FUNCTION_BLOCK MainStation EXTENDS TcoCore.TcoObject
VAR
    counter : INT;

    testAxis : AxisIaiLibrary.AxisIAI(THIS^, AxisLimits := AxisStats.AxisLimitsRfid);

    enable                 : BOOL := TRUE;
    controllWithCommActive : BOOL := TRUE;
    //Link this for example in Global to IN/Out
    gateWayStatus      : AxisIaiLibrary.GatewayStatus;
    gateWayControl     : AxisIaiLibrary.GatewayControl;
    DriveToPlcTestAxis : AxisIaiLibrary.PlcIn;
    PlcToDriveTestAxis : AxisIaiLibrary.PlcOut;
END_VAR

counter := counter + 1;

IF (THIS^.counter MOD 13 = 0) THEN
    THIS^.Messenger.Info('opalalla').Pin();
END_IF

IF (THIS^.counter MOD 400 = 0) THEN
    THIS^.Messenger.Error('ich Poste').Pin();
END_IF

testAxis
(
    inEnabled        := enable
    , GateWayStatus  := gateWayStatus
    , GateWayControl := gateWayControl
    , DriveToPlc     := DriveToPlcTestAxis
    , PlcToDrive     := PlcToDriveTestAxis
);

gateWayControl.GatewayControl0.MON := controllWithCommActive;

END_FUNCTION_BLOCK

(* stored: Version 1.1.0.1, ProductVersion 3.1.4024.12
   POU MainStation: Id {133c6404-7ee3-4d52-81ac-dadf34168d5f}, SpecialFunc None *)
